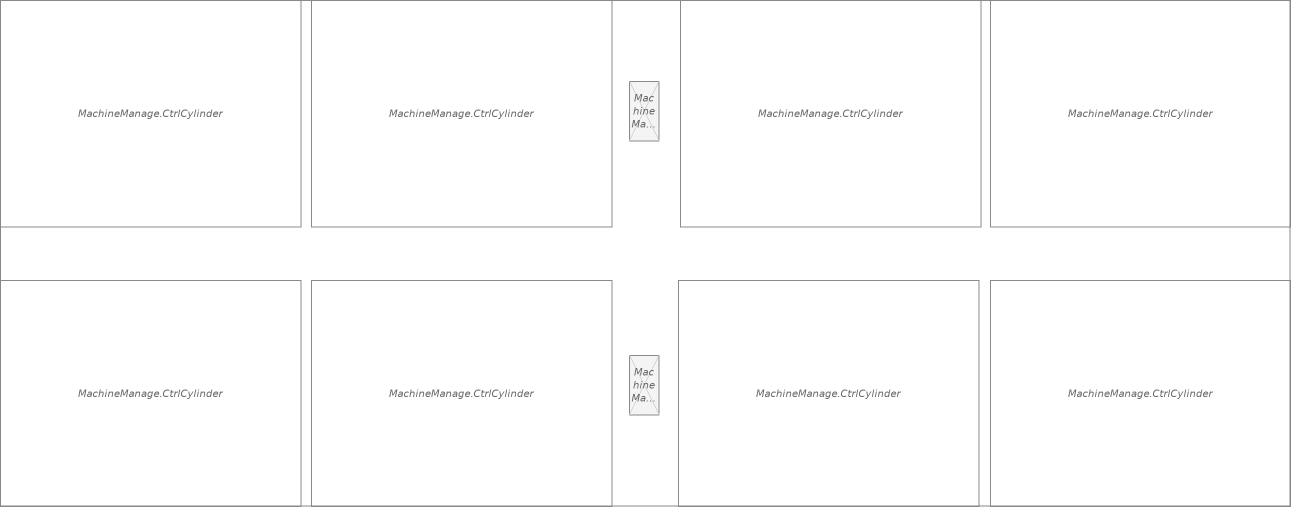
VISUALIZATION CtrlCylinder_Page  // 1291x507
VAR_INPUT
	System:				REFERENCE TO ST_System;
	Cylinder:			REFERENCE TO ARRAY[0..50] OF ST_Cylinder;
	CylinderData:		REFERENCE TO ARRAY[0..50] OF ST_CylinderData;
	Length:				INT;
END_VAR
VAR
	_i:					INT;
END_VAR
    Frame (0,0 301x227), invisible if: Length<=_i
        shows MachineManage.CtrlCylinder(System := System, Cylinder := Cylinder[_i], CylinderData := CylinderData[_i])
    Frame (311,0 301x227), invisible if: Length<=_i+1
        shows MachineManage.CtrlCylinder(System := System, Cylinder := Cylinder[_i+1], CylinderData := CylinderData[_i+1])
    Frame (0,280 301x227), invisible if: Length<=_i+2
        shows MachineManage.CtrlCylinder(System := System, Cylinder := Cylinder[_i+2], CylinderData := CylinderData[_i+2])
    Frame (311,280 301x227), invisible if: Length<=_i+3
        shows MachineManage.CtrlCylinder(System := System, Cylinder := Cylinder[_i+3], CylinderData := CylinderData[_i+3])
    Frame (680,0 301x227), invisible if: Length<=_i+4
        shows MachineManage.CtrlCylinder(System := System, Cylinder := Cylinder[_i+4], CylinderData := CylinderData[_i+4])
    Frame (678,280 301x227), invisible if: Length<=_i+6
        shows MachineManage.CtrlCylinder(System := System, Cylinder := Cylinder[_i+6], CylinderData := CylinderData[_i+6])
    Frame (990,0 301x227), invisible if: Length<=_i+5
        shows MachineManage.CtrlCylinder(System := System, Cylinder := Cylinder[_i+5], CylinderData := CylinderData[_i+5])
    Frame (990,280 301x227), invisible if: Length<=_i+7
        shows MachineManage.CtrlCylinder(System := System, Cylinder := Cylinder[_i+7], CylinderData := CylinderData[_i+7])
    Image (629,81 30x60), image: MachineManage.ImagePool.prev
        OnMouseDown: execute {
            IF _i-8>=0 THEN
            	_i:=_i-8;
            END_IF
        }
    Image (629,355 30x60), image: MachineManage.ImagePool.next
        OnMouseClick: execute {
            IF Length>_i+8 THEN
            	_i:=_i+8;
            END_IF
        }
END_VISUALIZATION

(* stored: Version 1.1.0.1, ProductVersion 3.1.4024.3
   Visu CtrlCylinder_Page: Id {bf29ba17-9d15-40fc-b516-34589c2be9a3} *)
